FUNCTION_BLOCK CollisionGroup IMPLEMENTS ICollisionGroup
VAR_INPUT
END_VAR
VAR_OUTPUT
END_VAR
VAR
	_caGroup : Tc3_McCoordinatedMotion.AXES_GROUP_REF;
	readStatus : Tc3_McCoordinatedMotion.MC_GroupReadStatus;
	resetCAGroup : ResetGroup(THIS^);
END_VAR

readStatus(
	AxesGroup:= _caGroup, 
	Enable:= TRUE );
resetCAGroup();

PROPERTY GroupRef : reference to AXES_GROUP_REF
GET
GroupRef REF= _caGroup;
END_GET
END_PROPERTY

PROPERTY GroupState : CAGroupStatus
GET
IF readStatus.GroupDisabled THEN
	GroupState := CAGroupStatus.mcGroupStateDisabled;
ELSIF readStatus.GroupErrorStop THEN
	GroupState := CAGroupStatus.mcGroupStateErrorStop;
ELSIF readStatus.GroupHoming THEN
	GroupState := CAGroupStatus.mcGroupStateHoming;
ELSIF readStatus.GroupMoving THEN
	GroupState := CAGroupStatus.mcGroupStateMoving;
ELSIF readStatus.GroupNotReady THEN
	GroupState := CAGroupStatus.mcGroupStateNotReady;
ELSIF readStatus.GroupStandby THEN
	GroupState := CAGroupStatus.mcGroupStateStandby;
ELSIF readStatus.GroupStopping THEN
	GroupState := CAGroupStatus.mcGroupStateStopping;
ELSIF readStatus.Error THEN
	GroupState := CAGroupStatus.mcGroupError;
END_IF
END_GET
END_PROPERTY

{warning 'add method implementation '}
METHOD Reset : BOOL
IF NOT resetCAGroup.Busy THEN
	resetCAGroup.Execute();
END_IF
END_METHOD

END_FUNCTION_BLOCK

(* stored: Version 1.1.0.1, ProductVersion 3.1.4024.9
   POU CollisionGroup: Id {0bc361f9-56cf-433c-aec7-a5801fd95d6e}, SpecialFunc None
   Property GroupRef: Id {6faf36db-c068-43d3-aa12-55d90013f979}
   Get Get: Id {c6dbe199-1644-405b-b519-b28e2b4f4703}
   Property GroupState: Id {eabcea1b-8fd2-4f17-a82d-d1eb5e302aca}
   Get Get: Id {e79d0405-66e0-4012-9a7b-d329b25966d5}
   Method Reset: Id {0ff9600a-32e3-414b-ae78-07f4f0e53dd3} *)
